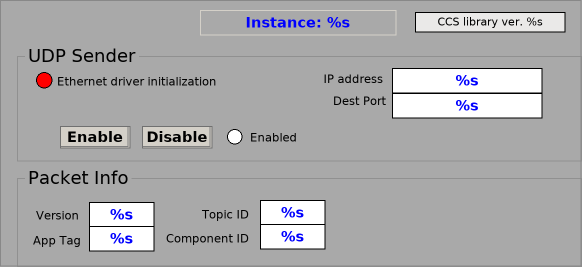
VISUALIZATION GUI_TEMPLATE_MUDPI_SENDER  // 582x267
VAR_INPUT
	m_DeviceName : STRING;
END_VAR
VAR_IN_OUT
	m_Instance : FB_MUDPI_SENDER;
END_VAR
    GroupBox (17,48 565x113), "UDP Sender"
        Rectangle (375,20 150x25), "%s", text variable: m_Instance._destinationIpAddressString
            OnMouseDown: write the text variable via Edit
        Label (285,18 84x26), "IP address"
        Label (37,19 240x29), "Ethernet driver initialization"
        Ellipse (19,24 16x16), tooltip "RED - False GREEN - True", colour toggle: m_Instance.bSuccessfulInitializationOfRealtimeDriver
        Label (265,40 107x26), "Dest Port"
        Rectangle (375,45 150x25), "%s", text variable: m_Instance._destinationPort
            OnMouseDown: write the text variable via Edit
        Button (43,78 70x22), "Enable", tooltip "Enable Diagnostics"
            OnMouseClick: execute { m_Instance.bEnableSending := TRUE; }
        Button (125,78 70x22), "Disable", tooltip "Disable Diagnostics"
            OnMouseClick: execute { m_Instance.bEnableSending := FALSE; }
        Label (230,75 61x29), "Enabled"
        Ellipse (210,81 15x15), tooltip "WHITE - Disabled GREEN - Enabled", colour toggle: m_Instance.bEnableSending
    Rectangle (200,10 196x25), "Instance: %s", text variable: m_Instance.instance_name
    Rectangle (415,12 150x20), "CCS library ver. %s", text variable: m_Instance.sLibVersion
    GroupBox (17,170 565x97), "Packet Info"
        Label (6,31 59x29), "Version"
        Label (6,56 61x29), "App Tag"
        Label (176,30 59x29), "Topic ID"
        Label (148,54 87x29), "Component ID"
        Rectangle (243,30 65x25), "%s", text variable: m_Instance.packet_info.topicId
            OnMouseDown: write the text variable via Edit
        Rectangle (243,54 65x25), "%s", text variable: m_Instance.packet_info.componentId
            OnMouseDown: write the text variable via Edit
        Rectangle (72,32 65x25), "%s", text variable: m_Instance.packet_info.version
            OnMouseDown: write the text variable via Edit
    Rectangle (89,226 65x25), "%s", text variable: m_Instance.packet_info.appTag
        OnMouseDown: write the text variable via Edit
END_VISUALIZATION

(* stored: Version 1.1.0.1, ProductVersion 3.1.4024.11
   Visu GUI_TEMPLATE_MUDPI_SENDER: Id {70e1fc48-d90b-4831-97ff-e2644e419c8c} *)
